{attribute 'GeneratedUsingTerminal: EPP7041-1002-0016'}
{attribute addProperty BoxType "EPP7041-1002-0016"}
{attribute addProperty Id "EnableBOOL1ResetBOOL1Reduce_torqueBOOL1Digital_output_1BOOL1"}
{attribute addProperty CRC "1607755581"}
{attribute addProperty Size "4"}
TYPE Control_5FD4673D :
STRUCT
	{attribute addProperty Name "Enable"}
	Enable : BOOL;
	{attribute addProperty Name "Reset"}
	Reset : BOOL;
	{attribute addProperty Name "Reduce_torque"}
	Reduce_torque : BOOL;
	{attribute addProperty Name "Digital_output_1"}
	Digital_output_1 : BOOL;
END_STRUCT
END_TYPE

(* stored: Version 1.2.0.0, ProductVersion 3.1.4024.9
   DUT Control_5FD4673D: Id {51b57ec7-b115-474f-94b0-44284dfe7cf9} *)
